{attribute addProperty BoxType "EL4021-0000-0016"}
{attribute addProperty Id "AO_OutputsAT %Q*AO_Outputs_F57FA4F91620WcStateAT %I*WcState_64F6A8C6810InfoDataAT %I*InfoData_BC63D37F80100"}
{attribute addProperty CRC "1748927295"}
{attribute addProperty SizeInBites "104"}
{attribute addProperty SizeInBytes "13"}
TYPE EL4021_A49381BF :
STRUCT
	{attribute addProperty Name "AO_Outputs"}
	AO_Outputs : AO_Outputs_F57FA4F9;
	{attribute addProperty Name "WcState"}
	WcState : WcState_64F6A8C6;
	{attribute addProperty Name "InfoData"}
	InfoData : InfoData_BC63D37F;
END_STRUCT
END_TYPE

(* stored: Version 1.2.0.0, ProductVersion 3.1.4024.9
   DUT EL4021_A49381BF: Id {dc1e618a-e720-4247-a3ee-7b126a9944bb} *)
